ABB RobotStudio station: Trainingai4.rsstnx

Station Trainingai4 (saved by RobotStudio 22.2.10013.1)
Controller Trainings5
  mechanical unit ROB_1: IRB4600_60_205_C_01, 6 joints, base frame (0, 0, 0) mm
Layout (positions relative to the parent item):
  - scGripper1 [smart component] at (-1960.6, -1054.25, 0) mm
      signals: DI diToolOpen, DI diToolClose, DO doToolOpened, DO doToolClosed, DO doPartPresent
      connections:
        LineSensor.SensorOut -> scGripper1.doPartPresent
        Detacher.Executed -> scGripper1.doToolOpened
        Attacher.Executed -> scGripper1.doToolClosed
        PoseMover.Executed -> Detacher.Execute
        PoseMover_2.Executed -> Attacher.Execute
        scGripper1.diToolOpen -> PoseMover.Execute
        scGripper1.diToolClose -> PoseMover_2.Execute
        LineSensor.SensedPart => Attacher.Child
        Attacher.Child => Detacher.Child
    - LineSensor [smart component, from Components\LineSensor.rslib] at (-7.15, -52.96, 0) mm
        properties: Start=[2.42780829058322 0.0931553945848375 0.59655]; End=[2.376167 0.062155 0.59655]; Radius=0.002; SensedPart=(none); SensedPoint=[0 0 0]
      - _sensorPart_ [part], size 53.7 x 34.4 x 4 mm
    - Attacher [smart component, from Components\Attacher.rslib]
        properties: Parent=(none); Flange=0; Child=(none); Mount=false; Offset=[0 0 0]; Orientation=[0 0 0]
    - Detacher [smart component, from Components\Detacher.rslib]
        properties: Child=(none); KeepPosition=true
    - PoseMover [smart component, from Components\PoseMover.rslib]
        properties: Mechanism=(none); Pose=0; Duration=1
    - PoseMover_2 [smart component, from Components\PoseMover.rslib]
        properties: Mechanism=(none); Pose=2; Duration=1
  - scGripper2 [smart component] at (570.25, 1720.75, 382.61) mm, rotated rx 0 ry 0 rz -63.28 deg
      properties: DetacherChild=(none)
      signals: DI diGripperOpen, DO doGripperOpened, DI diMagnetOn
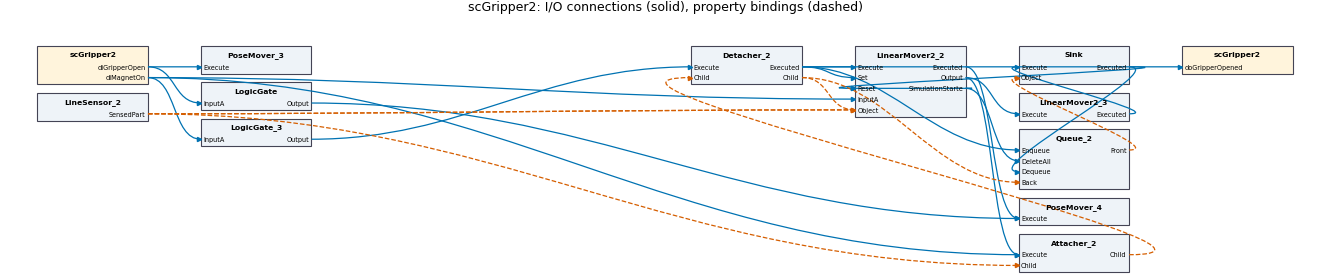
      connections:
        scGripper2.diGripperOpen -> PoseMover_3.Execute
        LinearMover2_2.Executed -> PoseMover_4.Execute
        Detacher_2.Executed -> LinearMover_2.Execute
        LinearMover2_3.Executed -> Sink.Execute
        Detacher_2.Executed -> LogicSRLatch.Set
        LogicSRLatch.Output -> LinearMover2_3.Execute
        Sink.Executed -> LogicSRLatch.Reset
        SimulationEvents_2.SimulationStarted -> LogicSRLatch.Reset
        Detacher_2.Executed -> Queue_2.Enqueue
        SimulationEvents_2.SimulationStarted -> Queue_2.DeleteAll
        Sink.Executed -> Queue_2.Dequeue
        Detacher_2.Executed -> scGripper2.doGripperOpened
        scGripper2.diGripperOpen -> LogicGate.InputA
        LogicGate.Output -> PoseMover_4.Execute
        scGripper2.diMagnetOn -> LogicGate_2.InputA
        LogicGate_2.Output -> Attacher_2.Execute
        scGripper2.diMagnetOn -> Attacher_2.Execute
        scGripper2.diMagnetOn -> LogicGate_3.InputA
        LogicGate_3.Output -> Detacher_2.Execute
        LineSensor_2.SensedPart => Attacher_2.Child
        Attacher_2.Child => Detacher_2.Child
        LineSensor_2.SensedPart => LinearMover2_2.Object
        LineSensor_2.SensedPart => Positioner_3.Object
        Detacher_2.Child => LinearMover_2.Object
        Detacher_2.Child => Queue_2.Back
        Queue_2.Front => Sink.Object
    - LineSensor_2 [smart component, from Components\LineSensor.rslib]
        properties: Start=[1.917656 0.079550000000004 0.234999999999997]; End=[1.917656 0.079550000000004 0.211400999999997]; Radius=0.002; SensedPart=(none); SensedPoint=[0 0 0]
      - _sensorPart_ [part], size 4 x 4 x 23.6 mm
    - PoseMover_3 [smart component, from Components\PoseMover.rslib]
        properties: Mechanism=tGripper2; Pose=2; Duration=0.5
    - PoseMover_4 [smart component, from Components\PoseMover.rslib]
        properties: Mechanism=tGripper2; Pose=0; Duration=0.5
    - Attacher_2 [smart component, from Components\Attacher.rslib]
        properties: Parent=IRB4600_60_205_C_01; Flange=0; Child=(none); Mount=false; Offset=[0 0 0]; Orientation=[0 0 0]
    - Detacher_2 [smart component, from Components\Detacher.rslib]
        properties: Child=(none); KeepPosition=true
    - LogicGate [smart component, from Components\LogicGate.rslib]
        properties: Operator=NOT; Delay=0
    - LogicGate_3 [smart component, from Components\LogicGate.rslib]
        properties: Operator=NOT; Delay=0
  - IRB4600_60_205_C_01 [mechanism] at (0, 0, 0) mm; joint values [0.0292, 0.4591, 0.0259, 0, 1.0857, -0.4372] (rad or m)
      links: Base, Link1, Link2, Link3, Link4, Link5, Link6
  - extHolder [mechanism] at (-1960.6, -1054.25, 0) mm; joint values [0] (rad or m)
      links: L1, Link
  - tGripper2 [mechanism] at (1504.07, 43.9, 874.01) mm, rotated rx -180 ry 0 rz -153.28 deg; joint values [1.5708, 1.5708, 1.5708, 1.5708] (rad or m)
      TCP tGripper2 at (0, 187, 0) mm, rotated rx 0 ry -90 rz -90 deg
      links: Baze, Kaire1, Kaire2, Desine1, Desine
  - tGripper1 [mechanism] at (204.61, -1164.7, 660) mm, rotated rx 180 ry 0 rz -150 deg; joint values [0, 0] (rad or m)
      TCP tGripper1 at (0, 85.55, -289) mm, rotated rx 180 ry 0 rz 90 deg
      links: Base, Kaire, Desine
  - scPalletConveyor [smart component]
      connections:
        Source.Executed -> LinearMover2.Execute
        Source.Executed -> Queue.Enqueue
        SimulationEvents.SimulationStarted -> Queue.DeleteAll
        SimulationEvents.SimulationStarted -> Source.Execute
        Source.Copy => LinearMover2.Object
        Source.Copy => Queue.Back
    - LinearMover2 [smart component, from Components\LinearMover2.rslib] at (-2600, 0, 0) mm
        properties: Object=scPalletWithParts_13; Direction=[-0.1 0 0]; Distance=2.6; Duration=5; Reference=Global; ReferenceObject=(none)
    - Source [smart component, from Components\Source.rslib] at (-2600, 0, 0) mm
        properties: Source=scPalletWithParts; Copy=scPalletWithParts_13; Parent=(none); Position=[0 0 0]; Orientation=[0 0 0]; Transient=false; PhysicsBehavior=0
    - scPalletWithParts [smart component] at (-4135.48, 0, -268.92) mm
        connections:
          ParametricBox.GeneratedPart => MatrixRepeater.Source
      - ParametricBox [smart component, from Components\ParametricBox.rslib] at (2772.59, 525, 316.05) mm
          properties: SizeX=0.5; SizeY=0.035; SizeZ=0.015; GeneratedPart=GeneratedPart; KeepGeometry=true
        - GeneratedPart [part], size 500 x 35 x 15 mm
      - MatrixRepeater [smart component, from Components\MatrixRepeater.rslib] at (2768.94, 525, 444) mm
          properties: Source=GeneratedPart; CountX=2; CountY=5; CountZ=1; OffsetX=0.6; OffsetY=0.2; OffsetZ=0.1
        - GeneratedPart [part], size 500 x 35 x 15 mm
        - GeneratedPart [part] at (600, 0, 0) mm, size 500 x 35 x 15 mm
        - GeneratedPart [part] at (0, 200, 0) mm, size 500 x 35 x 15 mm
        - GeneratedPart [part] at (600, 200, 0) mm, size 500 x 35 x 15 mm
        - GeneratedPart [part] at (0, 400, 0) mm, size 500 x 35 x 15 mm
        - GeneratedPart [part] at (600, 400, 0) mm, size 500 x 35 x 15 mm
        - GeneratedPart [part] at (0, 600, 0) mm, size 500 x 35 x 15 mm
        - GeneratedPart [part] at (600, 600, 0) mm, size 500 x 35 x 15 mm
        - GeneratedPart [part] at (0, 800, 0) mm, size 500 x 35 x 15 mm
        - GeneratedPart [part] at (600, 800, 0) mm, size 500 x 35 x 15 mm
      - Solid Face pallet [part] at (2668.87, 425, 300) mm, size 1300 x 1000 x 144 mm
    - Chain Conveyor [part] at (0, 525, 0) mm, size 4159.4 x 900 x 300 mm
    - SimulationEvents [smart component, from Components\SimulationEvents.rslib]
    - Queue [smart component, from Components\Queue.rslib]
        properties: Back=scPalletWithParts_13; Front=scPalletWithParts_13; Queue={def94a46-63ab-4a30-ae87-9a6eb517e7c9}; NumberOfObjects=1
    - scPalletWithParts_13 [smart component] at (-2600, 0, 0) mm
        connections:
          ParametricBox.GeneratedPart => MatrixRepeater.Source
      - ParametricBox [smart component, from Components\ParametricBox.rslib] at (2772.59, 525, 316.05) mm
          properties: SizeX=0.5; SizeY=0.035; SizeZ=0.015; GeneratedPart=GeneratedPart; KeepGeometry=true
        - GeneratedPart [part], size 500 x 35 x 15 mm
      - MatrixRepeater [smart component, from Components\MatrixRepeater.rslib] at (2768.94, 525, 444) mm
          properties: Source=GeneratedPart; CountX=2; CountY=5; CountZ=1; OffsetX=0.6; OffsetY=0.2; OffsetZ=0.1
        - GeneratedPart [part], size 500 x 35 x 15 mm
        - GeneratedPart [part] at (600, 0, 0) mm, size 500 x 35 x 15 mm
        - GeneratedPart [part] at (0, 200, 0) mm, size 500 x 35 x 15 mm
        - GeneratedPart [part] at (600, 200, 0) mm, size 500 x 35 x 15 mm
        - GeneratedPart [part] at (0, 400, 0) mm, size 500 x 35 x 15 mm
        - GeneratedPart [part] at (600, 400, 0) mm, size 500 x 35 x 15 mm
        - GeneratedPart [part] at (0, 600, 0) mm, size 500 x 35 x 15 mm
        - GeneratedPart [part] at (600, 600, 0) mm, size 500 x 35 x 15 mm
        - GeneratedPart [part] at (0, 800, 0) mm, size 500 x 35 x 15 mm
        - GeneratedPart [part] at (600, 800, 0) mm, size 500 x 35 x 15 mm
      - Solid Face pallet [part] at (2668.87, 425, 300) mm, size 1300 x 1000 x 144 mm
  - scPartConveyor [smart component]
      properties: DetacherChild=(none)
      signals: DI diGripperOpened
      connections:
        SimulationEvents_2.SimulationStarted -> Queue_2.DeleteAll
        LinearMover2_3.Executed -> Sink.Execute
        Sink.Executed -> Queue_2.Dequeue
        scPartConveyor.diGripperOpened -> Queue_2.Enqueue
        Timer.Output -> LinearMover2_3.Execute
        scPartConveyor.diGripperOpened -> Timer.Active
        scPartConveyor.diGripperOpened -> LinearMover2_3.Execute
        scPartConveyor.DetacherChild => Queue_2.Back
        Queue_2.Front => Sink.Object
    - Belt Conveyor [part] at (1257.28, -128.32, 0) mm, rotated rx 0 ry 0 rz -90 deg, size 5091 x 400 x 600 mm
    - Sink [smart component, from Components\Sink.rslib]
        properties: Object=(none)
    - Queue_2 [smart component, from Components\Queue.rslib]
        properties: Back=(none); Front=(none); Queue={2dc8e61b-ebec-44af-ad14-0ed559f0599e};{a771ce6e-0ae6-4e53-ab8f-f897429e7bdc};{55db3552-5567-4b7d-9fc8-0461d874dd02};{eca2981a-a2f0-4461-8ce5-34812ac5fa19};{0c85abd3-7812-48b3-ae52-80a0c9b890cb};{4e699870-b5d5-45c6-8165-44d45a72ec64};{717bbeb6-b8bc-4b00-a186-3d805d64528c};{651f6ac5-aea8-47f9-ae17-ed7998c333a4};{7c32ac3b-945e-400d-8ce3-24234b8ee495};{71834a44-749a-4cb6-8886-d85a4c408215};{7ab371d3-c5f9-41aa-aa14-6d825ef1be4f};{28583303-bd4f-4e9c-906b-fdd82cf9f385};{6c8c032e-3ace-4d8c-9ade-9f0e9220f704};{53d18044-a4a6-47e9-a2fd-a88179a397c4};{f98f4791-6472-4895-9234-1f3cf1dbf26f};{76240e30-d61d-432f-bdfa-ab9751f1b838};{3e2c236a-aa4f-4aca-a898-b86b4838ce87};{8efbb0bd-58a3-4156-8114-2d818540220e};{383bef30-bc5f-4f9a-83c2-b0e34f40491d};{85feea3d-e578-435b-8a0a-43b224609656};{7d6159f7-02fe-4613-abe4-c9ae4e2f11ab};{33503d57-5cf7-4ece-aeb4-f011f00fb54d};{af74fe30-0894-4f1b-9fbe-9a7e2716110b};{af57b412-42c3-4c7b-8199-7909dbcf08f4};{018e3041-176c-43ec-8c03-727afeb9b32d};{8be667fe-11ba-4109-9375-b98e5219bea1};{d23d0b7f-f891-4a8f-bfba-fc5707fab13a};{b891840e-4aac-46b0-8260-738cb80d5b75};{fa70ff57-8a2c-476f-9041-d0400eecf8eb};{9c520f9e-5298-43dc-b2a8-0cb615bae637};{60e750eb-7b52-474d-ae52-ff52f4173b29};{2e5c8f01-c4b5-456c-9932-b4f5dee0107b};{7cc00504-0dce-4288-9317-d0d6fe0c5c7c};{a5f28ec1-5dc2-4ed1-8193-ab70b21bbfdf};{ce9ec1a0-0e60-4302-a700-a5878b59edd3};{793488a4-99cf-42ff-aac9-6560d6ab3dd0};{78454220-a91c-468d-8c3c-db103b123668};{05bacae4-9263-4ba8-b032-70854a68714a};{bcc7de2b-fc59-4f15-89ab-b5e14cbe93ed};{9891b9ae-2fa4-4f68-964b-9ce407872076};{d7a565d5-c072-4b25-882f-d1a2a52e6e9c};{434aaa15-53f6-4512-a66b-7f3fe4fc45fe};{71fa1183-a7c1-4c06-a958-2085be59233c};{ee92a2f4-ddd4-4dd9-a94a-1fa7b2ea8aa9};{e9d00a95-32e3-485a-b503-9f73064d7dc6};{3cbd8215-6d0a-44fe-96ef-1986add50c42};{57ff91f2-0418-4f3d-a072-d27c6e0443a5};{a6f9d328-43d9-4753-a787-2e56ff4d3629};{353e8426-c6fe-4f15-b35b-50b5f885b2b0};{a50f6d1d-e2b8-404c-9dd8-50b2cbaf5305};{388b40b8-c995-48d4-b52d-113233b0e056};{6edbdafd-e9ec-4de0-8d17-490c81950243};{bdd515a6-c659-4542-afba-7f80a878ea6f};{7dba5a3f-8987-4bc8-ac31-969e188650cf};{de197d9a-2bf1-4685-9c4d-aabb2d0097c6};{8d97396d-6d16-465d-81a1-fc052d015174};{240d990e-038f-4ecc-8256-6e7bb5f8bec8};{fcafca83-c2aa-4a33-b7d5-ba0fdc46e004};{04eb8b1e-7c74-46b9-8734-7058114e5df0};{5b710989-514e-4d7a-b81b-72de4c0376f3};{77626a9d-f373-433c-a002-7fc1b27d7ed8};{e7fb0dd4-038f-4dd4-badc-155d66927d72};{87fc9cda-4f6e-44fa-b7ce-55f690ed2b64};{cf081dd7-6efd-4069-a464-6372a14ab6d3};{1dcbd514-ab29-42fb-a6f9-b7738e3fe18f};{7e055ee7-0bb8-4b19-aeae-7017d5662d06};{1a903323-41c6-4dfd-be20-7e9888df4bfb};{ab005678-ed27-4967-949f-ecc786924a2b};{095d61a3-3060-40a1-bd32-4be819dd842c};{927962db-11c6-499e-bbfa-c08fd1b03a11};{f17bbe06-97fc-4356-9d07-c1119bec4420};{1c2b368f-d9dd-4055-81b3-84e8fc9d758b};{72b7e295-ac51-4b04-abd7-5b676489df1c};{5a2c718f-610d-4225-bd56-6d0df54475db};{312de803-3f5d-4c00-8272-d9c3f53573e2};{c7af1266-0f19-4cdb-b741-5e372a020094};{cc5d6710-0141-457f-9462-e9feeee04ca5};{cefbf1fa-d663-46e0-a1fa-a3224f3b812b};{55060ab4-aeb4-4055-be77-df6de6529960};{80e64bfc-18ae-42bd-bebb-791938804c9b};{2876dd3d-53db-43e6-9b86-6361dd8b2537};{1195bc43-a2ff-414a-bc4e-aab0af6197c7};{8bd3f78f-b29b-45f3-b3e7-b9374d08a2da};{4c92dddf-96b5-49f8-9cbc-2f92ad07502a}; NumberOfObjects=1
    - LinearMover2_3 [smart component, from Components\LinearMover2.rslib]
        properties: Object=Queue_2; Direction=[0 -4.5 0]; Distance=4; Duration=5; Reference=Global; ReferenceObject=(none)
  - scToolChanger_4 [smart component] at (-218.13, -822.8, 1208.38) mm, rotated rx 0 ry 60 rz 26.72 deg
      signals: DI diAttachTool, DI diDetachTool
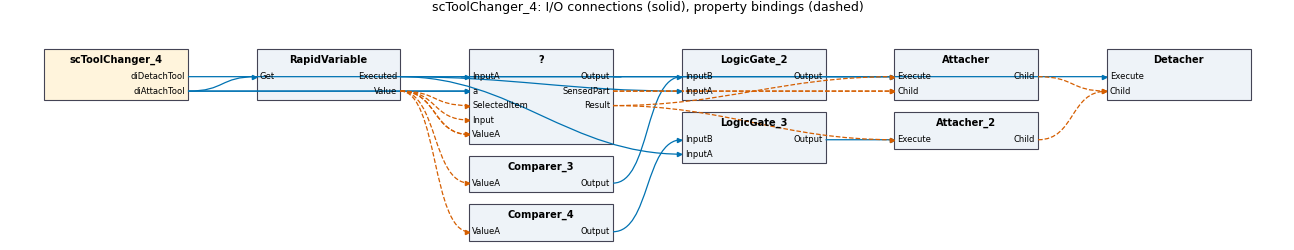
      connections:
        scToolChanger_4.diDetachTool -> Detacher.Execute
        scToolChanger_4.diAttachTool -> RapidVariable.Get
        ?.Output -> Attacher.Execute
        ?.Output -> ?.InputA
        scToolChanger_4.diAttachTool -> ?.a
        scToolChanger_4.diAttachTool -> ?.a
        Comparer_3.Output -> LogicGate_2.InputB
        LogicGate_2.Output -> Attacher.Execute
        Comparer_4.Output -> LogicGate_3.InputB
        LogicGate_3.Output -> Attacher_2.Execute
        RapidVariable.Executed -> LogicGate_3.InputA
        RapidVariable.Executed -> LogicGate_2.InputA
        ?.SensedPart => Attacher.Child
        Attacher.Child => Detacher.Child
        ?.SensedPart => Attacher.Child
        RapidVariable.Value => ?.SelectedItem
        RapidVariable.Value => ?.Input
        Attacher_2.Child => Detacher.Child
        RapidVariable.Value => ?.ValueA
        RapidVariable.Value => ?.ValueA
        ?.Result => Attacher.Execute
        ?.Result => Attacher_2.Execute
        RapidVariable.Value => Comparer_3.ValueA
        RapidVariable.Value => Comparer_4.ValueA
    - Swivel [part] at (1248.86, 0, 1502.5) mm, rotated rx 180 ry 60 rz 180 deg, size 181 x 209 x 109.7 mm
    - Attacher [smart component, from Components\Attacher.rslib]
        properties: Parent=IRB4600_60_205_C_01; Flange=0; Child=tGripper2; Mount=true; Offset=[0 0 0]; Orientation=[0 0 0]
    - Detacher [smart component, from Components\Detacher.rslib]
        properties: Child=tGripper1; KeepPosition=false
    - RapidVariable [smart component, from Components\RapidVariable.rslib]
        properties: DataType=num; Controller=Trainings5; Task=T_ROB1; Module=Main_; Variable=nWhichTool; Value=2
    - Attacher_2 [smart component, from Components\Attacher.rslib]
        properties: Parent=IRB4600_60_205_C_01; Flange=0; Child=tGripper1; Mount=true; Offset=[0 0 0]; Orientation=[0 0 0]
    - Comparer_3 [smart component, from Components\Comparer.rslib]
        properties: ValueA=2; Operator===; ValueB=2
    - Comparer_4 [smart component, from Components\Comparer.rslib]
        properties: ValueA=2; Operator===; ValueB=1
    - LogicGate_2 [smart component, from Components\LogicGate.rslib]
        properties: Operator=AND; Delay=0
    - LogicGate_3 [smart component, from Components\LogicGate.rslib]
        properties: Operator=AND; Delay=0
Attachment: scGripper1 is attached to tGripper1 / Base
Attachment: scGripper2 is attached to tGripper2 / Baze
Attachment: scToolChanger_4 is attached to IRB4600_60_205_C_01 / Link6
Attachment: tGripper2 is attached to IRB4600_60_205_C_01 / Link6
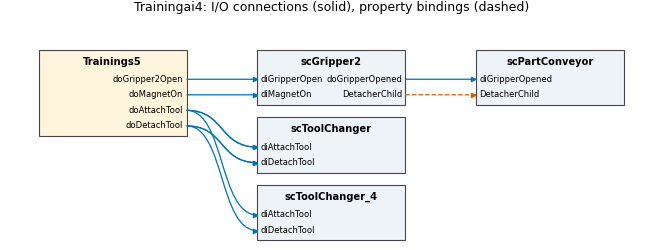
Station logic (signal -> signal, property => property):
  scGripper2.doGripperOpened -> scPartConveyor.diGripperOpened
  Trainings5.doGripper2Open -> scGripper2.diGripperOpen
  Trainings5.doMagnetOn -> scGripper2.diMagnetOn
  Trainings5.doAttachTool -> scToolChanger.diAttachTool
  Trainings5.doDetachTool -> scToolChanger.diDetachTool
  Trainings5.doAttachTool -> scToolChanger_3.diAttachTool
  Trainings5.doDetachTool -> scToolChanger_3.diDetachTool
  Trainings5.doAttachTool -> scToolChanger_4.diAttachTool
  Trainings5.doDetachTool -> scToolChanger_4.diDetachTool
  scGripper2.DetacherChild => scPartConveyor.DetacherChild
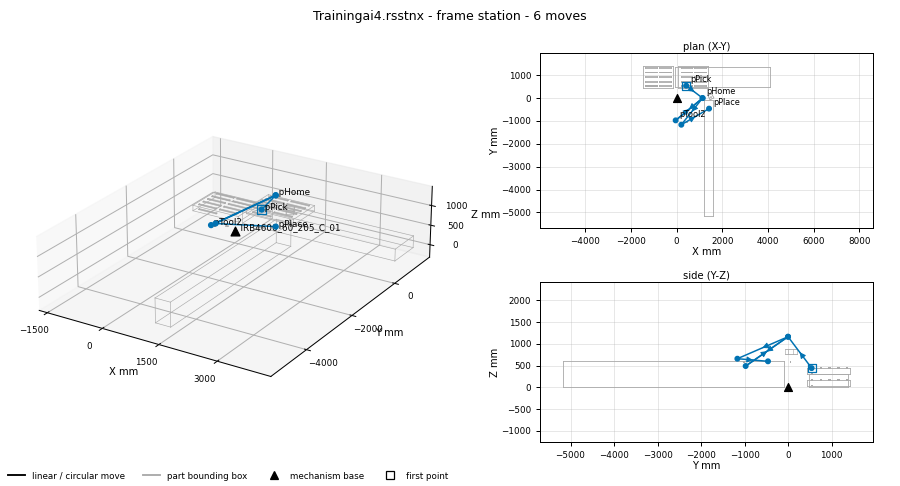
[picture p0: tool path of Trainingai4.rsstnx in frame station, 6 of 6 moves have a stored position in this frame; points joined in program order, loops and branches not executed]
Targets, tools, work objects and paths stored in the station, written as RAPID:
! task T_ROB1
MODULE CalibData
  PERS tooldata tGripper1:=[TRUE,[[-289,0,168.55],[1,0,0,0]],[5,[0,0,100],[1,0,0,0],0,0,0]];
  PERS tooldata tGripper2:=[TRUE,[[0,0,172.001],[1,0,0,0]],[3,[0,0,100],[1,0,0,0],0,0,0]];
ENDMODULE

! task T_ROB1
MODULE CalibData
  TASK PERS wobjdata wPallet:=[FALSE,TRUE,"",[[68.866,424.996,300],[1,0,0,0]],[[0,0,0],[1,0,0,0]]];
  CONST robtarget pPick:=[[350.075,117.5,144],[0,-0.707106781,0.707106781,0],[0,0,-1,0],[9E+09,9E+09,9E+09,9E+09,9E+09,9E+09]];
  CONST robtarget pHome:=[[1135,0,1165],[0,0,1,0],[0,0,0,0],[9E+09,9E+09,9E+09,9E+09,9E+09,9E+09]];
  CONST robtarget pPlace:=[[1417.902,-460.91,600],[0,0,1,0],[0,0,0,0],[9E+09,9E+09,9E+09,9E+09,9E+09,9E+09]];
  PROC Path_10()
    MoveL pPick,v1000,z100,tGripper2\WObj:=wPallet;
    MoveL pHome,v1000,z100,tGripper2\WObj:=wobj0;
    MoveL pTool2,v1000,z100,tool0\WObj:=wobj0;
    MoveL pHome,v1000,z100,tGripper2\WObj:=wobj0;
    MoveL pTool1,v1000,z100,tool0\WObj:=wobj0;
    MoveL pPlace,v1000,z100,tGripper2\WObj:=wobj0;
  ENDPROC
ENDMODULE

! task T_ROB1
MODULE Module1
  CONST robtarget pTool2:=[[-42.943005524,-974.204110584,491.401],[0,-0.707106781,0.707106781,0],[-2,0,-3,0],[9E+09,9E+09,9E+09,9E+09,9E+09,9E+09]];
  CONST robtarget pTool1:=[[204.606994476,-1164.704110584,660],[0,-0.258819045,0.965925826,0],[-1,0,-2,0],[9E+09,9E+09,9E+09,9E+09,9E+09,9E+09]];
ENDMODULE

! task T_ROB1
MODULE CalibDataR1
  PERS tooldata tGripper2:=[TRUE,[[0,0,270],[1,0,0,0]],[3,[0,0,100],[1,0,0,0],0,0,0]];
ENDMODULE

